FUNCTION_BLOCK ThreeConCtl (* Composite Function Block Type *)
  (* Standard: 61499-2 *)
  (* Version 0.2, 2003-12-05, JHC, Rockwell Automation, Renamed from NEWCOMPFB. *)
  (* Version 0.1, 2002-01-08, JHC, Rockwell Automation, Added DLY FB as example. *)
  (* Version 0.0, 2000-05-27, JHC, Rockwell Automation *)
  (* Compiler header: package fb.rt.cs725; *)
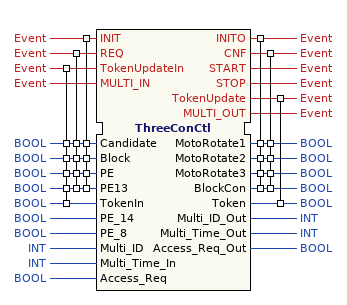
  EVENT_INPUT
    INIT WITH Candidate, Block, PE, PE13; (* Initialization Request *)
    REQ WITH Block, Candidate, PE, PE13; (* Normal Execution Request *)
    TokenUpdateIn WITH Candidate, Block, PE, PE13, TokenIn;
    MULTI_IN;
  END_EVENT
  EVENT_OUTPUT
    INITO WITH MotoRotate1, MotoRotate2, MotoRotate3, BlockCon; (* Initialization Confirm *)
    CNF WITH MotoRotate1, MotoRotate2, MotoRotate3, BlockCon; (* Execution Confirmation *)
    START;
    STOP;
    TokenUpdate WITH Token;
    MULTI_OUT;
  END_EVENT
  VAR_INPUT
    Candidate : BOOL;
    Block : BOOL;
    PE : BOOL;
    PE13 : BOOL;
    TokenIn : BOOL;
    PE_14 : BOOL;
    PE_8 : BOOL;
    Multi_ID : INT;
    Multi_Time_In : INT;
    Access_Req : BOOL;
  END_VAR
  VAR_OUTPUT
    MotoRotate1 : BOOL;
    MotoRotate2 : BOOL;
    MotoRotate3 : BOOL;
    BlockCon : BOOL;
    Token : BOOL;
    Multi_ID_Out : INT;
    Multi_Time_Out : INT;
    Access_Req_Out : BOOL;
  END_VAR
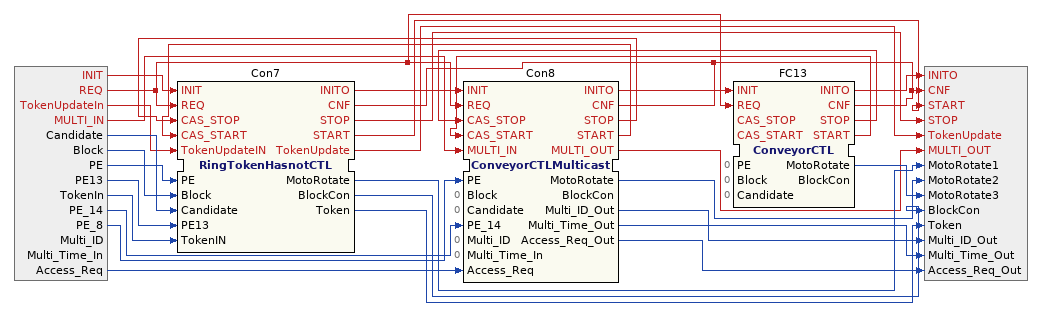
  FBS
    Con7 : RingTokenHasnotCTL;
    Con8 : ConveyorCTLMulticast(Block := 0, Candidate := 0, Multi_ID := 0, Multi_Time_In := 0);
    FC13 : ConveyorCTL(PE := 0, Block := 0, Candidate := 0);
  END_FBS
  EVENT_CONNECTIONS
    INIT TO Con7.INIT;
    REQ TO Con7.REQ;
    Con7.INITO TO Con8.INIT;
    Con8.INITO TO FC13.INIT;
    FC13.INITO TO INITO;
    FC13.CNF TO CNF;
    REQ TO Con8.REQ;
    REQ TO FC13.REQ;
    Con7.CNF TO CNF;
    Con8.CNF TO CNF;
    TokenUpdateIn TO Con7.TokenUpdateIN;
    Con7.TokenUpdate TO TokenUpdate;
    MULTI_IN TO Con8.MULTI_IN;
    Con8.MULTI_OUT TO MULTI_OUT;
    FC13.START TO Con8.CAS_START;
    FC13.STOP TO Con8.CAS_STOP;
    Con8.START TO Con7.CAS_START;
    Con8.STOP TO Con7.CAS_STOP;
    Con7.STOP TO STOP;
    Con7.START TO START;
  END_CONNECTIONS
  DATA_CONNECTIONS
    FC13.MotoRotate TO MotoRotate3;
    Con8.MotoRotate TO MotoRotate2;
    Con7.MotoRotate TO MotoRotate1;
    PE TO Con7.PE;
    Block TO Con7.Block;
    Con7.BlockCon TO BlockCon;
    Candidate TO Con7.Candidate;
    PE13 TO Con7.PE13;
    TokenIn TO Con7.TokenIN;
    Con7.Token TO Token;
    PE_8 TO Con8.PE;
    Con8.Multi_ID_Out TO Multi_ID_Out;
    Con8.Multi_Time_Out TO Multi_Time_Out;
    Con8.Access_Req_Out TO Access_Req_Out;
    PE_14 TO Con8.PE_14;
    Access_Req TO Con8.Access_Req;
  END_CONNECTIONS
END_FUNCTION_BLOCK
